VISUALIZATION SingleFixture_1  // 1120x220
END_VISUALIZATION

(* stored: Version 1.1.0.1, ProductVersion 3.1.4024.12
   Visu SingleFixture_1: Id {645db971-9934-4260-ad90-c8fd8c0af206} *)
